PROGRAM MAIN
VAR
END_VAR

END_PROGRAM

(* stored: Version 1.1.0.1
   POU MAIN: Id {d8ec20df-8949-402c-85bd-d17a6cfdae81} *)
